ABB RobotStudio station: ABBPaintRobot.rspag

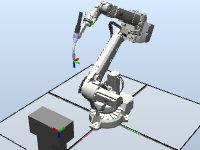
--- station ---
Station ABBPaintRobot (saved by RobotStudio 6.8.8148.134)
Controller IRB_2600ID_8kg_2.00m
  mechanical unit ROB_1: IRB2600ID_8_200__02, 6 joints, base frame (0, 0, 0) mm
Layout (positions relative to the parent item):
  - IRB2600ID_8_200__02 [mechanism, from Robots\IRB2600ID_8_200_G_02.rslib] at (0, 0, 0) mm; joint values [0, -0.957, 0.4843, 0, 1.1459, 0] (rad or m)
  - Binzel_air_22 [mechanism, from Tools\Binzel_air_22.rslib] at (337.53, 0, 1399.27) mm, rotated rx 180 ry 51.43 rz 180 deg
  - Part_1 [part] at (953.78, 0, 190.26) mm
  - Part_2 [part] at (953.94, -93.96, 490.36) mm
Attachment: Binzel_air_22 is attached to IRB2600ID_8_200__02 / Link6
Targets, tools, work objects and paths stored in the station and not in the controller backup, written as RAPID:
! task T_ROB1
MODULE Module1
  CONST robtarget Target_10:=[[1060.139962435,99.723394802,660.032584238],[0.005005717,0.000000004,-0.999987471,0.000000001],[0,-1,0,0],[9E+09,9E+09,9E+09,9E+09,9E+09,9E+09]];
  CONST robtarget Target_20:=[[204.629025164,93.494499262,29.906548442],[0.707097925,-0.003539557,0.003539553,0.707097919],[0,-1,0,0],[9E+09,9E+09,9E+09,9E+09,9E+09,9E+09]];
  PROC EX_PAINT()
    ConfL \Off;
    MoveJ create_robtarget(tgPos{1}),v100,z0,tWeldGun\WObj:=Workobject;
    MoveJ create_robtarget(tgPos{i}),v100,z0,tWeldGun\WObj:=Workobject;
    MoveJ pHome,v600,z10,tWeldGun\WObj:=wobj0;
  ENDPROC
  PROC Path_10()
    MoveL Target_10,v1000,z100,tWeldGun\WObj:=wobj0;
    MoveL Target_20,v1000,z100,tWeldGun\WObj:=Workobject;
    MoveL Target_20,v1000,z100,tWeldGun\WObj:=Workobject;
  ENDPROC
ENDMODULE


--- Backups/IRB_2600ID_8kg_2.00m/RAPID/TASK1/PROGMOD/CalibData.mod ---
MODULE CalibData
	PERS tooldata tWeldGun:=[TRUE,[[125.800591275,0,391.268161315],[0.898794046,0,0.438371147,0]],[3,[0,0,100],[0,1,0,0],0,0,0]];
	TASK PERS wobjdata Workobject:=[FALSE,TRUE,"",[[1153.634449017,304.352418096,689.939187119],[0,-0.707106781,0.707106781,0]],[[0,0,0],[1,0,0,0]]];
ENDMODULE

--- Backups/IRB_2600ID_8kg_2.00m/RAPID/TASK1/PROGMOD/Module1.mod ---
MODULE Module1

    CONST num STOP_PROC:=-1;
    CONST num TO_PAINT := 1;
    CONST num TO_WAIT := 0;
    VAR num flag:=0;
    PERS pos tgPos{500};
    VAR num targetsNum;
    VAR bool repeat := TRUE;
    CONST robtarget pHome:=[[564.982678405,0,1056.955004785],[0.0050058,0,-0.999987471,0],[0,0,0,0],[9E+09,9E+09,9E+09,9E+09,9E+09,9E+09]];


    PROC Main()

        targetsNum := 0;
        repeat := TRUE;
        flag := 0;

        WHILE flag>STOP_PROC DO
            IF flag=TO_PAINT THEN
                PAINT;
            ENDIF
            WaitTime 0.2;
        ENDWHILE


    ENDPROC

    FUNC robtarget Create_robtarget(pos position)
       RETURN [position,[0.707097925,-0.003539557,0.003539553,0.707097919],[0,-1,0,0],[9E9,9E9,9E9,9E9,9E9,9E9]];
    ENDFUNC

	PROC PAINT()

        VAR num i := 2;
        ConfL \Off;

        MoveJ create_robtarget(tgPos{1}),v100,z0,tWeldGun\WObj:=Workobject;

        WHILE repeat DO

            MoveJ create_robtarget(tgPos{i}),v100,z0,tWeldGun\WObj:=Workobject;
            i := i + 1;
            IF i > targetsNum THEN repeat := FALSE; ENDIF

        ENDWHILE

        flag := TO_WAIT;
        repeat := TRUE;

        MoveJ pHome,v600,z10,tWeldGun\WObj:=wobj0;

	ENDPROC

ENDMODULE
